// TIA Portal V15.1 export
// export: Created 2024-05-17T05:39:00.2667194Z, ExportSetting WithDefaults, DisplayName Totally Integrated Automation Portal, DisplayVersion V15.1 Update 5, DisplayName TIA Portal Openness, DisplayVersion V15.1 Update 5, DisplayName SINAMICS Startdrive Advanced, DisplayVersion V15.1, DisplayName G130, G150, S120, S150, SINAMICS MV, S210, DisplayVersion V15.1, DisplayName G110M, G120, G120C, G120D, G120P, DisplayVersion V15.1, DisplayName STEP 7 Professional, DisplayVersion V15.1 Update 5, DisplayName STEP 7 Safety, DisplayVersion V15.1, DisplayName WinCC Professional, DisplayVersion V15.1 Update 5, DisplayName SIMATIC Visualization Architect, DisplayVersion V15.1
FUNCTION "209000NCP01AK" : Void   // FC254, FBD
TITLE = 209000NCP01AK
{ S7_Optimized_Access := 'FALSE' }
AUTHOR : VCC
NAME : LocFnc
VERSION : 0.1
// stored: AutoNumber false, IsIECCheckEnabled false, SetENOAutomatically False, UDAEnableTagReadback false
   VAR_OUTPUT
      O_AlarmA : Bool;   // Alarm A
      O_AlarmB : Bool;   // Alarm B
      O_AlarmC : Bool;   // Alarm C
      O_AlarmD : Bool;   // Alarm D
      O_AlarmABCondition : Bool;   // Alarms resetable
      H_IAnim : Word;   // For animation of icon
   END_VAR
BEGIN

REGION Network 1: **** --------------------- AK01 --------------------- ****
END_REGION

REGION Network 2: **** 2.2 Alarms - Alarm generation **** AK01E1QM1 - AE01 EG1 - Overload protection power supply 24VDC
   // AE01 EG1 - Overload protection power supply 24VDC
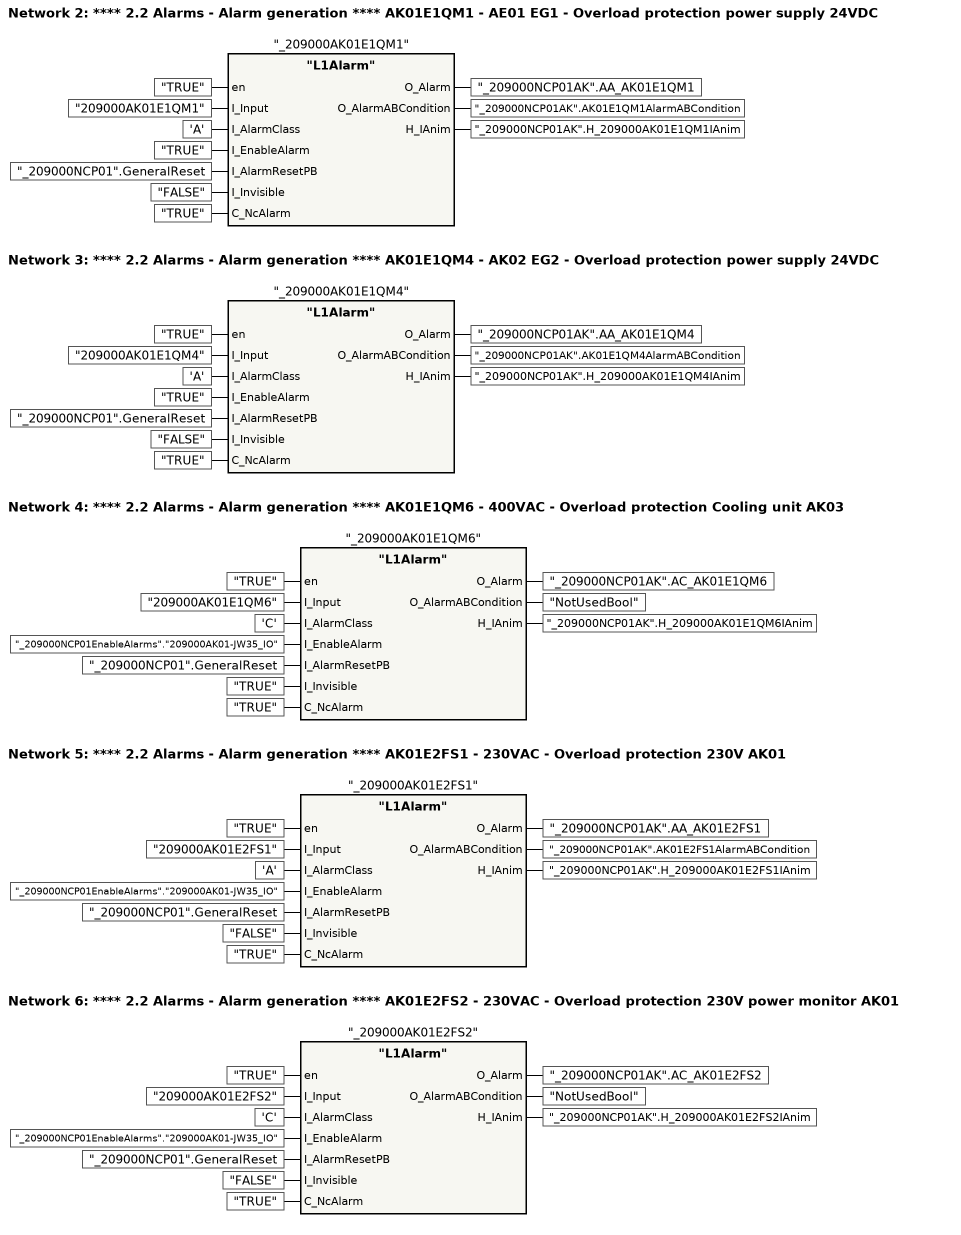
   IF "TRUE" THEN
       "_209000AK01E1QM1"(I_Input := "209000AK01E1QM1",   // "L1Alarm"
                          I_AlarmClass := 'A',
                          I_EnableAlarm := "TRUE",
                          I_AlarmResetPB := "_209000NCP01".GeneralReset,
                          I_Invisible := "FALSE",
                          C_NcAlarm := "TRUE",
                          O_Alarm => "_209000NCP01AK".AA_AK01E1QM1,
                          O_AlarmABCondition => "_209000NCP01AK".AK01E1QM1AlarmABCondition,
                          H_IAnim => "_209000NCP01AK".H_209000AK01E1QM1IAnim);
   END_IF;
END_REGION

REGION Network 3: **** 2.2 Alarms - Alarm generation **** AK01E1QM4 - AK02 EG2 - Overload protection power supply 24VDC
   // AK02 EG2 - Overload protection power supply 24VDC
   IF "TRUE" THEN
       "_209000AK01E1QM4"(I_Input := "209000AK01E1QM4",   // "L1Alarm"
                          I_AlarmClass := 'A',
                          I_EnableAlarm := "TRUE",
                          I_AlarmResetPB := "_209000NCP01".GeneralReset,
                          I_Invisible := "FALSE",
                          C_NcAlarm := "TRUE",
                          O_Alarm => "_209000NCP01AK".AA_AK01E1QM4,
                          O_AlarmABCondition => "_209000NCP01AK".AK01E1QM4AlarmABCondition,
                          H_IAnim => "_209000NCP01AK".H_209000AK01E1QM4IAnim);
   END_IF;
END_REGION

REGION Network 4: **** 2.2 Alarms - Alarm generation **** AK01E1QM6 - 400VAC - Overload protection Cooling unit AK03
   // 400VAC - Overload protection Cooling unit AK03
   IF "TRUE" THEN
       "_209000AK01E1QM6"(I_Input := "209000AK01E1QM6",   // "L1Alarm"
                          I_AlarmClass := 'C',
                          I_EnableAlarm := "_209000NCP01EnableAlarms"."209000AK01-JW35_IO",
                          I_AlarmResetPB := "_209000NCP01".GeneralReset,
                          I_Invisible := "TRUE",
                          C_NcAlarm := "TRUE",
                          O_Alarm => "_209000NCP01AK".AC_AK01E1QM6,
                          O_AlarmABCondition => "NotUsedBool",
                          H_IAnim => "_209000NCP01AK".H_209000AK01E1QM6IAnim);
   END_IF;
END_REGION

REGION Network 5: **** 2.2 Alarms - Alarm generation **** AK01E2FS1 - 230VAC - Overload protection 230V AK01
   // 230VAC - Overload protection 230V AK01
   IF "TRUE" THEN
       "_209000AK01E2FS1"(I_Input := "209000AK01E2FS1",   // "L1Alarm"
                          I_AlarmClass := 'A',
                          I_EnableAlarm := "_209000NCP01EnableAlarms"."209000AK01-JW35_IO",
                          I_AlarmResetPB := "_209000NCP01".GeneralReset,
                          I_Invisible := "FALSE",
                          C_NcAlarm := "TRUE",
                          O_Alarm => "_209000NCP01AK".AA_AK01E2FS1,
                          O_AlarmABCondition => "_209000NCP01AK".AK01E2FS1AlarmABCondition,
                          H_IAnim => "_209000NCP01AK".H_209000AK01E2FS1IAnim);
   END_IF;
END_REGION

REGION Network 6: **** 2.2 Alarms - Alarm generation **** AK01E2FS2 - 230VAC - Overload protection 230V power monitor AK01
   // 230VAC - Overload protection 230V power monitor AK01
   IF "TRUE" THEN
       "_209000AK01E2FS2"(I_Input := "209000AK01E2FS2",   // "L1Alarm"
                          I_AlarmClass := 'C',
                          I_EnableAlarm := "_209000NCP01EnableAlarms"."209000AK01-JW35_IO",
                          I_AlarmResetPB := "_209000NCP01".GeneralReset,
                          I_Invisible := "FALSE",
                          C_NcAlarm := "TRUE",
                          O_Alarm => "_209000NCP01AK".AC_AK01E2FS2,
                          O_AlarmABCondition => "NotUsedBool",
                          H_IAnim => "_209000NCP01AK".H_209000AK01E2FS2IAnim);
   END_IF;
END_REGION

REGION Network 7: **** 2.2 Alarms - Alarm generation **** AK01E2FS3 - 230VAC - Overload protection Socket + Light AK01-04
   // 230VAC - Overload protection Socket + Light AK01-04
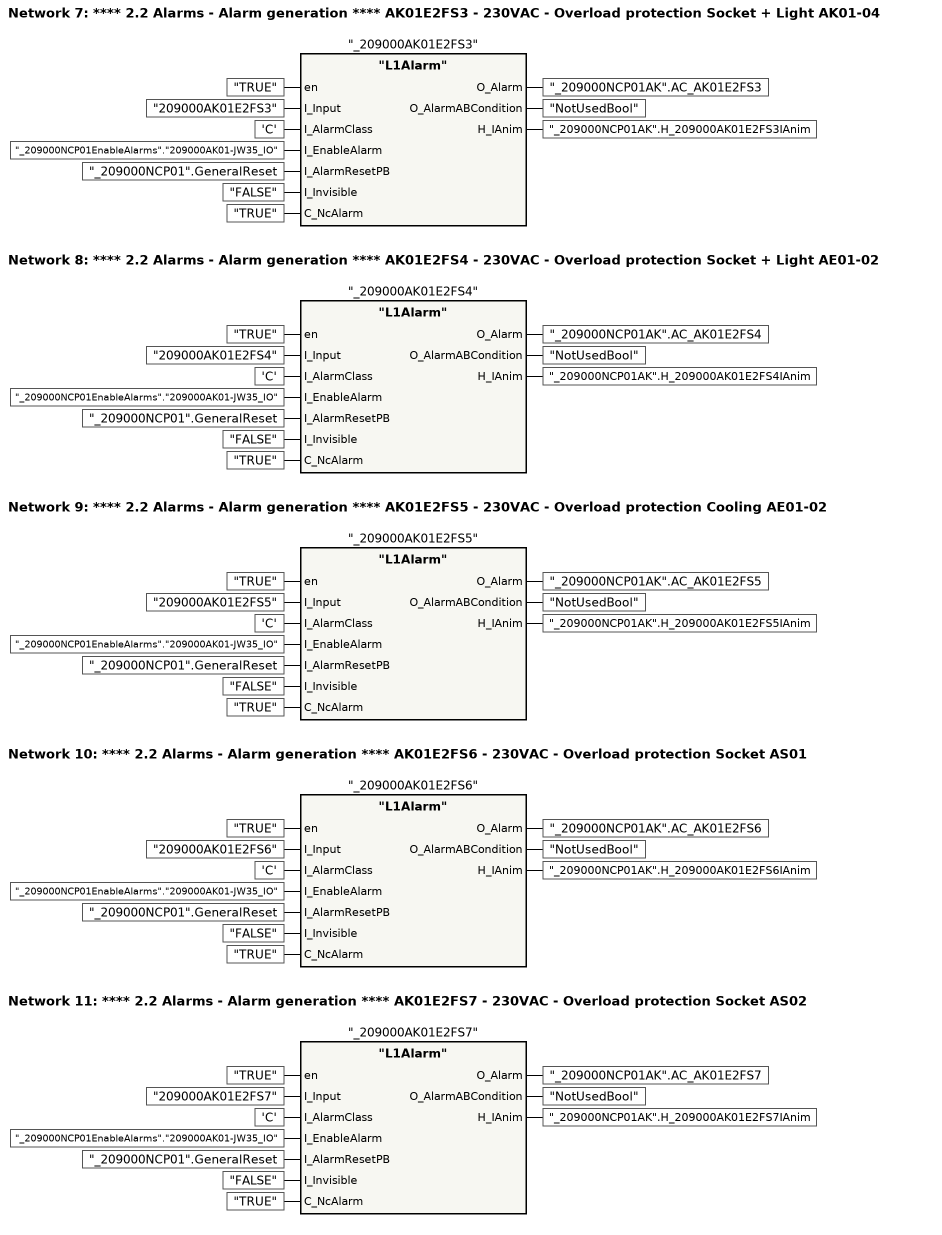
   IF "TRUE" THEN
       "_209000AK01E2FS3"(I_Input := "209000AK01E2FS3",   // "L1Alarm"
                          I_AlarmClass := 'C',
                          I_EnableAlarm := "_209000NCP01EnableAlarms"."209000AK01-JW35_IO",
                          I_AlarmResetPB := "_209000NCP01".GeneralReset,
                          I_Invisible := "FALSE",
                          C_NcAlarm := "TRUE",
                          O_Alarm => "_209000NCP01AK".AC_AK01E2FS3,
                          O_AlarmABCondition => "NotUsedBool",
                          H_IAnim => "_209000NCP01AK".H_209000AK01E2FS3IAnim);
   END_IF;
END_REGION

REGION Network 8: **** 2.2 Alarms - Alarm generation **** AK01E2FS4 - 230VAC - Overload protection Socket + Light AE01-02
   // 230VAC - Overload protection Socket + Light AE01-02
   IF "TRUE" THEN
       "_209000AK01E2FS4"(I_Input := "209000AK01E2FS4",   // "L1Alarm"
                          I_AlarmClass := 'C',
                          I_EnableAlarm := "_209000NCP01EnableAlarms"."209000AK01-JW35_IO",
                          I_AlarmResetPB := "_209000NCP01".GeneralReset,
                          I_Invisible := "FALSE",
                          C_NcAlarm := "TRUE",
                          O_Alarm => "_209000NCP01AK".AC_AK01E2FS4,
                          O_AlarmABCondition => "NotUsedBool",
                          H_IAnim => "_209000NCP01AK".H_209000AK01E2FS4IAnim);
   END_IF;
END_REGION

REGION Network 9: **** 2.2 Alarms - Alarm generation **** AK01E2FS5 - 230VAC - Overload protection Cooling AE01-02
   // 230VAC - Overload protection Cooling AE01-02
   IF "TRUE" THEN
       "_209000AK01E2FS5"(I_Input := "209000AK01E2FS5",   // "L1Alarm"
                          I_AlarmClass := 'C',
                          I_EnableAlarm := "_209000NCP01EnableAlarms"."209000AK01-JW35_IO",
                          I_AlarmResetPB := "_209000NCP01".GeneralReset,
                          I_Invisible := "FALSE",
                          C_NcAlarm := "TRUE",
                          O_Alarm => "_209000NCP01AK".AC_AK01E2FS5,
                          O_AlarmABCondition => "NotUsedBool",
                          H_IAnim => "_209000NCP01AK".H_209000AK01E2FS5IAnim);
   END_IF;
END_REGION

REGION Network 10: **** 2.2 Alarms - Alarm generation **** AK01E2FS6 - 230VAC - Overload protection Socket AS01
   // 230VAC - Overload protection Socket AS01
   IF "TRUE" THEN
       "_209000AK01E2FS6"(I_Input := "209000AK01E2FS6",   // "L1Alarm"
                          I_AlarmClass := 'C',
                          I_EnableAlarm := "_209000NCP01EnableAlarms"."209000AK01-JW35_IO",
                          I_AlarmResetPB := "_209000NCP01".GeneralReset,
                          I_Invisible := "FALSE",
                          C_NcAlarm := "TRUE",
                          O_Alarm => "_209000NCP01AK".AC_AK01E2FS6,
                          O_AlarmABCondition => "NotUsedBool",
                          H_IAnim => "_209000NCP01AK".H_209000AK01E2FS6IAnim);
   END_IF;
END_REGION

REGION Network 11: **** 2.2 Alarms - Alarm generation **** AK01E2FS7 - 230VAC - Overload protection Socket AS02
   // 230VAC - Overload protection Socket AS02
   IF "TRUE" THEN
       "_209000AK01E2FS7"(I_Input := "209000AK01E2FS7",   // "L1Alarm"
                          I_AlarmClass := 'C',
                          I_EnableAlarm := "_209000NCP01EnableAlarms"."209000AK01-JW35_IO",
                          I_AlarmResetPB := "_209000NCP01".GeneralReset,
                          I_Invisible := "FALSE",
                          C_NcAlarm := "TRUE",
                          O_Alarm => "_209000NCP01AK".AC_AK01E2FS7,
                          O_AlarmABCondition => "NotUsedBool",
                          H_IAnim => "_209000NCP01AK".H_209000AK01E2FS7IAnim);
   END_IF;
END_REGION

REGION Network 12: **** 2.2 Alarms - Alarm generation **** AK01E1FV1 - Surge protection 400VAC AK01 NOK
   // Surge protection 400VAC AK01 NOK
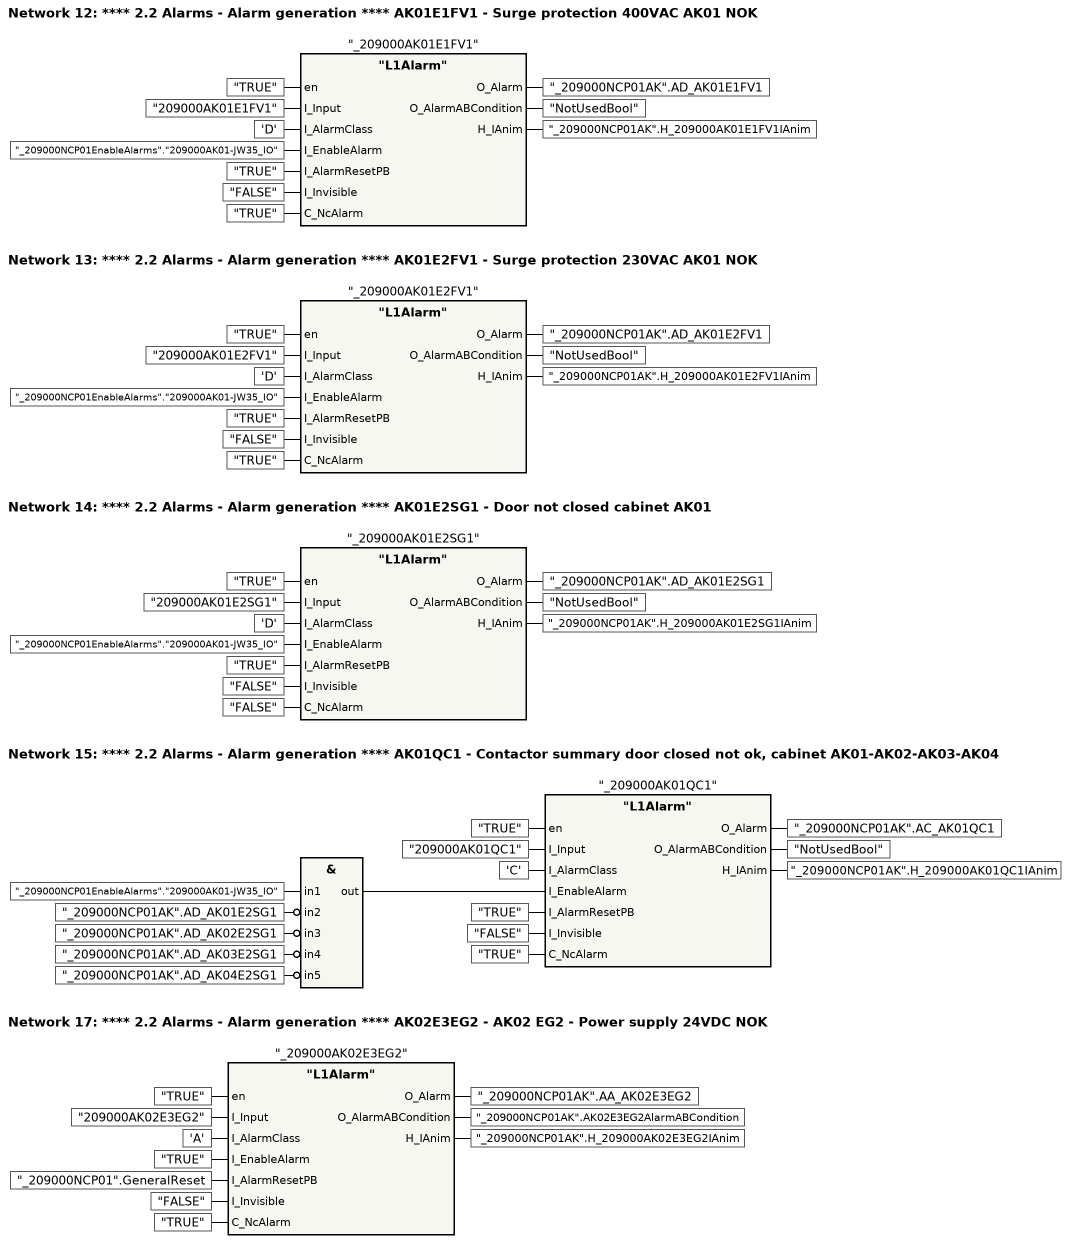
   IF "TRUE" THEN
       "_209000AK01E1FV1"(I_Input := "209000AK01E1FV1",   // "L1Alarm"
                          I_AlarmClass := 'D',
                          I_EnableAlarm := "_209000NCP01EnableAlarms"."209000AK01-JW35_IO",
                          I_AlarmResetPB := "TRUE",
                          I_Invisible := "FALSE",
                          C_NcAlarm := "TRUE",
                          O_Alarm => "_209000NCP01AK".AD_AK01E1FV1,
                          O_AlarmABCondition => "NotUsedBool",
                          H_IAnim => "_209000NCP01AK".H_209000AK01E1FV1IAnim);
   END_IF;
END_REGION

REGION Network 13: **** 2.2 Alarms - Alarm generation **** AK01E2FV1 - Surge protection 230VAC AK01 NOK
   // Surge protection 230VAC AK01 NOK
   IF "TRUE" THEN
       "_209000AK01E2FV1"(I_Input := "209000AK01E2FV1",   // "L1Alarm"
                          I_AlarmClass := 'D',
                          I_EnableAlarm := "_209000NCP01EnableAlarms"."209000AK01-JW35_IO",
                          I_AlarmResetPB := "TRUE",
                          I_Invisible := "FALSE",
                          C_NcAlarm := "TRUE",
                          O_Alarm => "_209000NCP01AK".AD_AK01E2FV1,
                          O_AlarmABCondition => "NotUsedBool",
                          H_IAnim => "_209000NCP01AK".H_209000AK01E2FV1IAnim);
   END_IF;
END_REGION

REGION Network 14: **** 2.2 Alarms - Alarm generation **** AK01E2SG1 - Door not closed cabinet AK01
   // Door not closed cabinet AK01
   IF "TRUE" THEN
       "_209000AK01E2SG1"(I_Input := "209000AK01E2SG1",   // "L1Alarm"
                          I_AlarmClass := 'D',
                          I_EnableAlarm := "_209000NCP01EnableAlarms"."209000AK01-JW35_IO",
                          I_AlarmResetPB := "TRUE",
                          I_Invisible := "FALSE",
                          C_NcAlarm := "FALSE",
                          O_Alarm => "_209000NCP01AK".AD_AK01E2SG1,
                          O_AlarmABCondition => "NotUsedBool",
                          H_IAnim => "_209000NCP01AK".H_209000AK01E2SG1IAnim);
   END_IF;
END_REGION

REGION Network 15: **** 2.2 Alarms - Alarm generation **** AK01QC1 - Contactor summary door closed not ok, cabinet AK01-AK02-AK03-AK04
   // Contactor summary door closed not ok, cabinet AK01-AK02-AK03-AK04
   IF "TRUE" THEN
       "_209000AK01QC1"(I_Input := "209000AK01QC1",   // "L1Alarm"
                        I_AlarmClass := 'C',
                        I_EnableAlarm := "_209000NCP01EnableAlarms"."209000AK01-JW35_IO" AND NOT "_209000NCP01AK".AD_AK01E2SG1 AND NOT "_209000NCP01AK".AD_AK02E2SG1 AND NOT "_209000NCP01AK".AD_AK03E2SG1 AND NOT "_209000NCP01AK".AD_AK04E2SG1,
                        I_AlarmResetPB := "TRUE",
                        I_Invisible := "FALSE",
                        C_NcAlarm := "TRUE",
                        O_Alarm => "_209000NCP01AK".AC_AK01QC1,
                        O_AlarmABCondition => "NotUsedBool",
                        H_IAnim => "_209000NCP01AK".H_209000AK01QC1IAnim);
   END_IF;
END_REGION

REGION Network 16: **** --------------------- AK02 --------------------- ****
END_REGION

REGION Network 17: **** 2.2 Alarms - Alarm generation **** AK02E3EG2 - AK02 EG2 - Power supply 24VDC NOK
   // AK02 EG2 - Power supply 24VDC NOK
   IF "TRUE" THEN
       "_209000AK02E3EG2"(I_Input := "209000AK02E3EG2",   // "L1Alarm"
                          I_AlarmClass := 'A',
                          I_EnableAlarm := "TRUE",
                          I_AlarmResetPB := "_209000NCP01".GeneralReset,
                          I_Invisible := "FALSE",
                          C_NcAlarm := "TRUE",
                          O_Alarm => "_209000NCP01AK".AA_AK02E3EG2,
                          O_AlarmABCondition => "_209000NCP01AK".AK02E3EG2AlarmABCondition,
                          H_IAnim => "_209000NCP01AK".H_209000AK02E3EG2IAnim);
   END_IF;
END_REGION

REGION Network 18: **** 2.2 Alarms - Alarm generation **** AK02E3FV2 - AK02 EG2 - Surge protection 24VDC NOK
   // AK02 EG2 - Surge protection 24VDC NOK
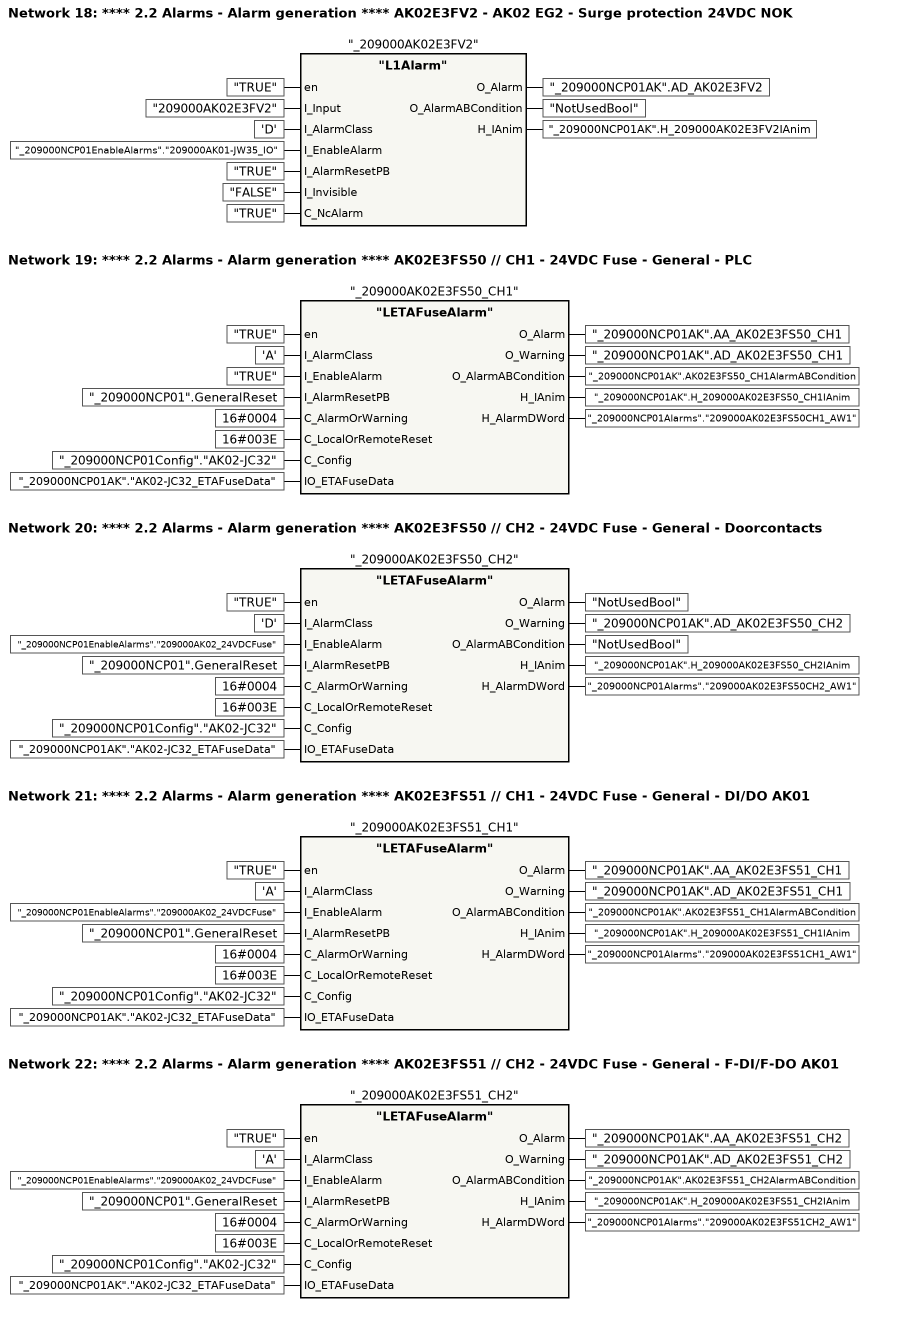
   IF "TRUE" THEN
       "_209000AK02E3FV2"(I_Input := "209000AK02E3FV2",   // "L1Alarm"
                          I_AlarmClass := 'D',
                          I_EnableAlarm := "_209000NCP01EnableAlarms"."209000AK01-JW35_IO",
                          I_AlarmResetPB := "TRUE",
                          I_Invisible := "FALSE",
                          C_NcAlarm := "TRUE",
                          O_Alarm => "_209000NCP01AK".AD_AK02E3FV2,
                          O_AlarmABCondition => "NotUsedBool",
                          H_IAnim => "_209000NCP01AK".H_209000AK02E3FV2IAnim);
   END_IF;
END_REGION

REGION Network 19: **** 2.2 Alarms - Alarm generation **** AK02E3FS50 // CH1 - 24VDC Fuse - General - PLC
   // 24VDC Fuse - General - PLC
   IF "TRUE" THEN
       "_209000AK02E3FS50_CH1"(I_AlarmClass := 'A',   // "LETAFuseAlarm"
                               I_EnableAlarm := "TRUE",
                               I_AlarmResetPB := "_209000NCP01".GeneralReset,
                               C_AlarmOrWarning := 16#0004,
                               C_LocalOrRemoteReset := 16#003E,
                               C_Config := "_209000NCP01Config"."AK02-JC32",
                               IO_ETAFuseData := "_209000NCP01AK"."AK02-JC32_ETAFuseData",
                               O_Alarm => "_209000NCP01AK".AA_AK02E3FS50_CH1,
                               O_Warning => "_209000NCP01AK".AD_AK02E3FS50_CH1,
                               O_AlarmABCondition => "_209000NCP01AK".AK02E3FS50_CH1AlarmABCondition,
                               H_IAnim => "_209000NCP01AK".H_209000AK02E3FS50_CH1IAnim,
                               H_AlarmDWord => "_209000NCP01Alarms"."209000AK02E3FS50CH1_AW1");
   END_IF;
END_REGION

REGION Network 20: **** 2.2 Alarms - Alarm generation **** AK02E3FS50 // CH2 - 24VDC Fuse - General - Doorcontacts
   // 24VDC Fuse - General - Doorcontacts
   IF "TRUE" THEN
       "_209000AK02E3FS50_CH2"(I_AlarmClass := 'D',   // "LETAFuseAlarm"
                               I_EnableAlarm := "_209000NCP01EnableAlarms"."209000AK02_24VDCFuse",
                               I_AlarmResetPB := "_209000NCP01".GeneralReset,
                               C_AlarmOrWarning := 16#0004,
                               C_LocalOrRemoteReset := 16#003E,
                               C_Config := "_209000NCP01Config"."AK02-JC32",
                               IO_ETAFuseData := "_209000NCP01AK"."AK02-JC32_ETAFuseData",
                               O_Alarm => "NotUsedBool",
                               O_Warning => "_209000NCP01AK".AD_AK02E3FS50_CH2,
                               O_AlarmABCondition => "NotUsedBool",
                               H_IAnim => "_209000NCP01AK".H_209000AK02E3FS50_CH2IAnim,
                               H_AlarmDWord => "_209000NCP01Alarms"."209000AK02E3FS50CH2_AW1");
   END_IF;
END_REGION

REGION Network 21: **** 2.2 Alarms - Alarm generation **** AK02E3FS51 // CH1 - 24VDC Fuse - General - DI/DO AK01
   // 24VDC Fuse - General - DI/DO AK01
   IF "TRUE" THEN
       "_209000AK02E3FS51_CH1"(I_AlarmClass := 'A',   // "LETAFuseAlarm"
                               I_EnableAlarm := "_209000NCP01EnableAlarms"."209000AK02_24VDCFuse",
                               I_AlarmResetPB := "_209000NCP01".GeneralReset,
                               C_AlarmOrWarning := 16#0004,
                               C_LocalOrRemoteReset := 16#003E,
                               C_Config := "_209000NCP01Config"."AK02-JC32",
                               IO_ETAFuseData := "_209000NCP01AK"."AK02-JC32_ETAFuseData",
                               O_Alarm => "_209000NCP01AK".AA_AK02E3FS51_CH1,
                               O_Warning => "_209000NCP01AK".AD_AK02E3FS51_CH1,
                               O_AlarmABCondition => "_209000NCP01AK".AK02E3FS51_CH1AlarmABCondition,
                               H_IAnim => "_209000NCP01AK".H_209000AK02E3FS51_CH1IAnim,
                               H_AlarmDWord => "_209000NCP01Alarms"."209000AK02E3FS51CH1_AW1");
   END_IF;
END_REGION

REGION Network 22: **** 2.2 Alarms - Alarm generation **** AK02E3FS51 // CH2 - 24VDC Fuse - General - F-DI/F-DO AK01
   // 24VDC Fuse - General - F-DI/F-DO AK01
   IF "TRUE" THEN
       "_209000AK02E3FS51_CH2"(I_AlarmClass := 'A',   // "LETAFuseAlarm"
                               I_EnableAlarm := "_209000NCP01EnableAlarms"."209000AK02_24VDCFuse",
                               I_AlarmResetPB := "_209000NCP01".GeneralReset,
                               C_AlarmOrWarning := 16#0004,
                               C_LocalOrRemoteReset := 16#003E,
                               C_Config := "_209000NCP01Config"."AK02-JC32",
                               IO_ETAFuseData := "_209000NCP01AK"."AK02-JC32_ETAFuseData",
                               O_Alarm => "_209000NCP01AK".AA_AK02E3FS51_CH2,
                               O_Warning => "_209000NCP01AK".AD_AK02E3FS51_CH2,
                               O_AlarmABCondition => "_209000NCP01AK".AK02E3FS51_CH2AlarmABCondition,
                               H_IAnim => "_209000NCP01AK".H_209000AK02E3FS51_CH2IAnim,
                               H_AlarmDWord => "_209000NCP01Alarms"."209000AK02E3FS51CH2_AW1");
   END_IF;
END_REGION

REGION Network 23: **** 2.2 Alarms - Alarm generation **** AK02E3FS52 // CH1 - 24VDC Fuse - General - DI/DO AK03
   // 24VDC Fuse - General - DI/DO AK03
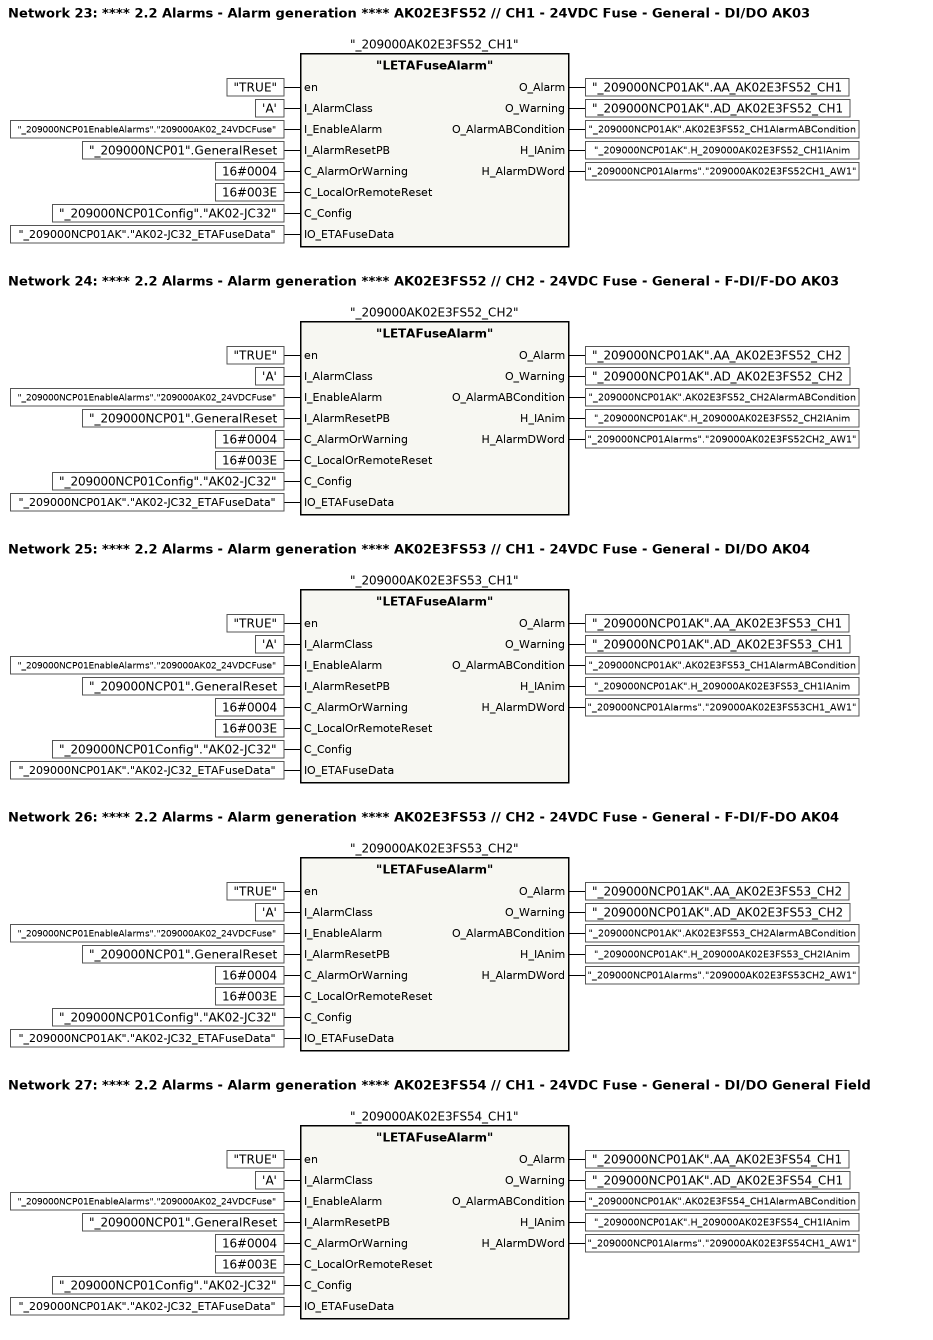
   IF "TRUE" THEN
       "_209000AK02E3FS52_CH1"(I_AlarmClass := 'A',   // "LETAFuseAlarm"
                               I_EnableAlarm := "_209000NCP01EnableAlarms"."209000AK02_24VDCFuse",
                               I_AlarmResetPB := "_209000NCP01".GeneralReset,
                               C_AlarmOrWarning := 16#0004,
                               C_LocalOrRemoteReset := 16#003E,
                               C_Config := "_209000NCP01Config"."AK02-JC32",
                               IO_ETAFuseData := "_209000NCP01AK"."AK02-JC32_ETAFuseData",
                               O_Alarm => "_209000NCP01AK".AA_AK02E3FS52_CH1,
                               O_Warning => "_209000NCP01AK".AD_AK02E3FS52_CH1,
                               O_AlarmABCondition => "_209000NCP01AK".AK02E3FS52_CH1AlarmABCondition,
                               H_IAnim => "_209000NCP01AK".H_209000AK02E3FS52_CH1IAnim,
                               H_AlarmDWord => "_209000NCP01Alarms"."209000AK02E3FS52CH1_AW1");
   END_IF;
END_REGION

REGION Network 24: **** 2.2 Alarms - Alarm generation **** AK02E3FS52 // CH2 - 24VDC Fuse - General - F-DI/F-DO AK03
   // 24VDC Fuse - General - F-DI/F-DO AK03
   IF "TRUE" THEN
       "_209000AK02E3FS52_CH2"(I_AlarmClass := 'A',   // "LETAFuseAlarm"
                               I_EnableAlarm := "_209000NCP01EnableAlarms"."209000AK02_24VDCFuse",
                               I_AlarmResetPB := "_209000NCP01".GeneralReset,
                               C_AlarmOrWarning := 16#0004,
                               C_LocalOrRemoteReset := 16#003E,
                               C_Config := "_209000NCP01Config"."AK02-JC32",
                               IO_ETAFuseData := "_209000NCP01AK"."AK02-JC32_ETAFuseData",
                               O_Alarm => "_209000NCP01AK".AA_AK02E3FS52_CH2,
                               O_Warning => "_209000NCP01AK".AD_AK02E3FS52_CH2,
                               O_AlarmABCondition => "_209000NCP01AK".AK02E3FS52_CH2AlarmABCondition,
                               H_IAnim => "_209000NCP01AK".H_209000AK02E3FS52_CH2IAnim,
                               H_AlarmDWord => "_209000NCP01Alarms"."209000AK02E3FS52CH2_AW1");
   END_IF;
END_REGION

REGION Network 25: **** 2.2 Alarms - Alarm generation **** AK02E3FS53 // CH1 - 24VDC Fuse - General - DI/DO AK04
   // 24VDC Fuse - General - DI/DO AK04
   IF "TRUE" THEN
       "_209000AK02E3FS53_CH1"(I_AlarmClass := 'A',   // "LETAFuseAlarm"
                               I_EnableAlarm := "_209000NCP01EnableAlarms"."209000AK02_24VDCFuse",
                               I_AlarmResetPB := "_209000NCP01".GeneralReset,
                               C_AlarmOrWarning := 16#0004,
                               C_LocalOrRemoteReset := 16#003E,
                               C_Config := "_209000NCP01Config"."AK02-JC32",
                               IO_ETAFuseData := "_209000NCP01AK"."AK02-JC32_ETAFuseData",
                               O_Alarm => "_209000NCP01AK".AA_AK02E3FS53_CH1,
                               O_Warning => "_209000NCP01AK".AD_AK02E3FS53_CH1,
                               O_AlarmABCondition => "_209000NCP01AK".AK02E3FS53_CH1AlarmABCondition,
                               H_IAnim => "_209000NCP01AK".H_209000AK02E3FS53_CH1IAnim,
                               H_AlarmDWord => "_209000NCP01Alarms"."209000AK02E3FS53CH1_AW1");
   END_IF;
END_REGION

REGION Network 26: **** 2.2 Alarms - Alarm generation **** AK02E3FS53 // CH2 - 24VDC Fuse - General - F-DI/F-DO AK04
   // 24VDC Fuse - General - F-DI/F-DO AK04
   IF "TRUE" THEN
       "_209000AK02E3FS53_CH2"(I_AlarmClass := 'A',   // "LETAFuseAlarm"
                               I_EnableAlarm := "_209000NCP01EnableAlarms"."209000AK02_24VDCFuse",
                               I_AlarmResetPB := "_209000NCP01".GeneralReset,
                               C_AlarmOrWarning := 16#0004,
                               C_LocalOrRemoteReset := 16#003E,
                               C_Config := "_209000NCP01Config"."AK02-JC32",
                               IO_ETAFuseData := "_209000NCP01AK"."AK02-JC32_ETAFuseData",
                               O_Alarm => "_209000NCP01AK".AA_AK02E3FS53_CH2,
                               O_Warning => "_209000NCP01AK".AD_AK02E3FS53_CH2,
                               O_AlarmABCondition => "_209000NCP01AK".AK02E3FS53_CH2AlarmABCondition,
                               H_IAnim => "_209000NCP01AK".H_209000AK02E3FS53_CH2IAnim,
                               H_AlarmDWord => "_209000NCP01Alarms"."209000AK02E3FS53CH2_AW1");
   END_IF;
END_REGION

REGION Network 27: **** 2.2 Alarms - Alarm generation **** AK02E3FS54 // CH1 - 24VDC Fuse - General - DI/DO General Field
   // 24VDC Fuse - General - DI/DO General Field
   IF "TRUE" THEN
       "_209000AK02E3FS54_CH1"(I_AlarmClass := 'A',   // "LETAFuseAlarm"
                               I_EnableAlarm := "_209000NCP01EnableAlarms"."209000AK02_24VDCFuse",
                               I_AlarmResetPB := "_209000NCP01".GeneralReset,
                               C_AlarmOrWarning := 16#0004,
                               C_LocalOrRemoteReset := 16#003E,
                               C_Config := "_209000NCP01Config"."AK02-JC32",
                               IO_ETAFuseData := "_209000NCP01AK"."AK02-JC32_ETAFuseData",
                               O_Alarm => "_209000NCP01AK".AA_AK02E3FS54_CH1,
                               O_Warning => "_209000NCP01AK".AD_AK02E3FS54_CH1,
                               O_AlarmABCondition => "_209000NCP01AK".AK02E3FS54_CH1AlarmABCondition,
                               H_IAnim => "_209000NCP01AK".H_209000AK02E3FS54_CH1IAnim,
                               H_AlarmDWord => "_209000NCP01Alarms"."209000AK02E3FS54CH1_AW1");
   END_IF;
END_REGION

REGION Network 28: **** 2.2 Alarms - Alarm generation **** AK02E3FS54 // CH2 - 24VDC Fuse - General - F-DI/F-DO General Field
   // 24VDC Fuse - General - F-DI/F-DO General Field
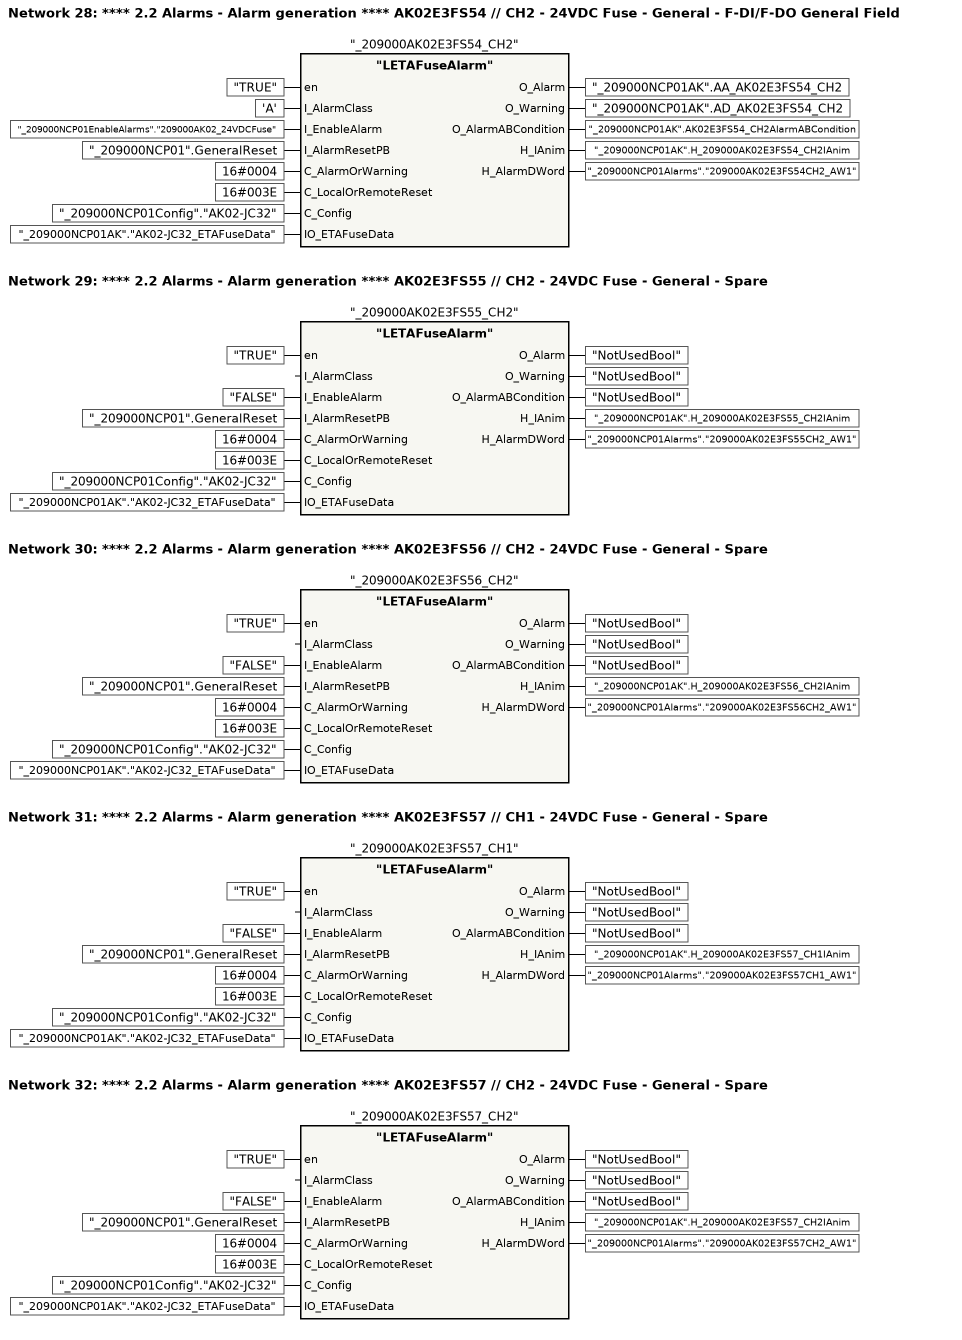
   IF "TRUE" THEN
       "_209000AK02E3FS54_CH2"(I_AlarmClass := 'A',   // "LETAFuseAlarm"
                               I_EnableAlarm := "_209000NCP01EnableAlarms"."209000AK02_24VDCFuse",
                               I_AlarmResetPB := "_209000NCP01".GeneralReset,
                               C_AlarmOrWarning := 16#0004,
                               C_LocalOrRemoteReset := 16#003E,
                               C_Config := "_209000NCP01Config"."AK02-JC32",
                               IO_ETAFuseData := "_209000NCP01AK"."AK02-JC32_ETAFuseData",
                               O_Alarm => "_209000NCP01AK".AA_AK02E3FS54_CH2,
                               O_Warning => "_209000NCP01AK".AD_AK02E3FS54_CH2,
                               O_AlarmABCondition => "_209000NCP01AK".AK02E3FS54_CH2AlarmABCondition,
                               H_IAnim => "_209000NCP01AK".H_209000AK02E3FS54_CH2IAnim,
                               H_AlarmDWord => "_209000NCP01Alarms"."209000AK02E3FS54CH2_AW1");
   END_IF;
END_REGION

REGION Network 29: **** 2.2 Alarms - Alarm generation **** AK02E3FS55 // CH2 - 24VDC Fuse - General - Spare
   // 24VDC Fuse - General - Spare
   IF "TRUE" THEN
       "_209000AK02E3FS55_CH2"(I_EnableAlarm := "FALSE",   // "LETAFuseAlarm"
                               I_AlarmResetPB := "_209000NCP01".GeneralReset,
                               C_AlarmOrWarning := 16#0004,
                               C_LocalOrRemoteReset := 16#003E,
                               C_Config := "_209000NCP01Config"."AK02-JC32",
                               IO_ETAFuseData := "_209000NCP01AK"."AK02-JC32_ETAFuseData",
                               O_Alarm => "NotUsedBool",
                               O_Warning => "NotUsedBool",
                               O_AlarmABCondition => "NotUsedBool",
                               H_IAnim => "_209000NCP01AK".H_209000AK02E3FS55_CH2IAnim,
                               H_AlarmDWord => "_209000NCP01Alarms"."209000AK02E3FS55CH2_AW1");
   END_IF;
END_REGION

REGION Network 30: **** 2.2 Alarms - Alarm generation **** AK02E3FS56 // CH2 - 24VDC Fuse - General - Spare
   // 24VDC Fuse - General - Spare
   IF "TRUE" THEN
       "_209000AK02E3FS56_CH2"(I_EnableAlarm := "FALSE",   // "LETAFuseAlarm"
                               I_AlarmResetPB := "_209000NCP01".GeneralReset,
                               C_AlarmOrWarning := 16#0004,
                               C_LocalOrRemoteReset := 16#003E,
                               C_Config := "_209000NCP01Config"."AK02-JC32",
                               IO_ETAFuseData := "_209000NCP01AK"."AK02-JC32_ETAFuseData",
                               O_Alarm => "NotUsedBool",
                               O_Warning => "NotUsedBool",
                               O_AlarmABCondition => "NotUsedBool",
                               H_IAnim => "_209000NCP01AK".H_209000AK02E3FS56_CH2IAnim,
                               H_AlarmDWord => "_209000NCP01Alarms"."209000AK02E3FS56CH2_AW1");
   END_IF;
END_REGION

REGION Network 31: **** 2.2 Alarms - Alarm generation **** AK02E3FS57 // CH1 - 24VDC Fuse - General - Spare
   // 24VDC Fuse - General - Spare
   IF "TRUE" THEN
       "_209000AK02E3FS57_CH1"(I_EnableAlarm := "FALSE",   // "LETAFuseAlarm"
                               I_AlarmResetPB := "_209000NCP01".GeneralReset,
                               C_AlarmOrWarning := 16#0004,
                               C_LocalOrRemoteReset := 16#003E,
                               C_Config := "_209000NCP01Config"."AK02-JC32",
                               IO_ETAFuseData := "_209000NCP01AK"."AK02-JC32_ETAFuseData",
                               O_Alarm => "NotUsedBool",
                               O_Warning => "NotUsedBool",
                               O_AlarmABCondition => "NotUsedBool",
                               H_IAnim => "_209000NCP01AK".H_209000AK02E3FS57_CH1IAnim,
                               H_AlarmDWord => "_209000NCP01Alarms"."209000AK02E3FS57CH1_AW1");
   END_IF;
END_REGION

REGION Network 32: **** 2.2 Alarms - Alarm generation **** AK02E3FS57 // CH2 - 24VDC Fuse - General - Spare
   // 24VDC Fuse - General - Spare
   IF "TRUE" THEN
       "_209000AK02E3FS57_CH2"(I_EnableAlarm := "FALSE",   // "LETAFuseAlarm"
                               I_AlarmResetPB := "_209000NCP01".GeneralReset,
                               C_AlarmOrWarning := 16#0004,
                               C_LocalOrRemoteReset := 16#003E,
                               C_Config := "_209000NCP01Config"."AK02-JC32",
                               IO_ETAFuseData := "_209000NCP01AK"."AK02-JC32_ETAFuseData",
                               O_Alarm => "NotUsedBool",
                               O_Warning => "NotUsedBool",
                               O_AlarmABCondition => "NotUsedBool",
                               H_IAnim => "_209000NCP01AK".H_209000AK02E3FS57_CH2IAnim,
                               H_AlarmDWord => "_209000NCP01Alarms"."209000AK02E3FS57CH2_AW1");
   END_IF;
END_REGION

REGION Network 33: **** 2.2 Alarms - Alarm generation **** AK02E2SG1 - Door not closed cabinet AK02
   // Door not closed cabinet AK02
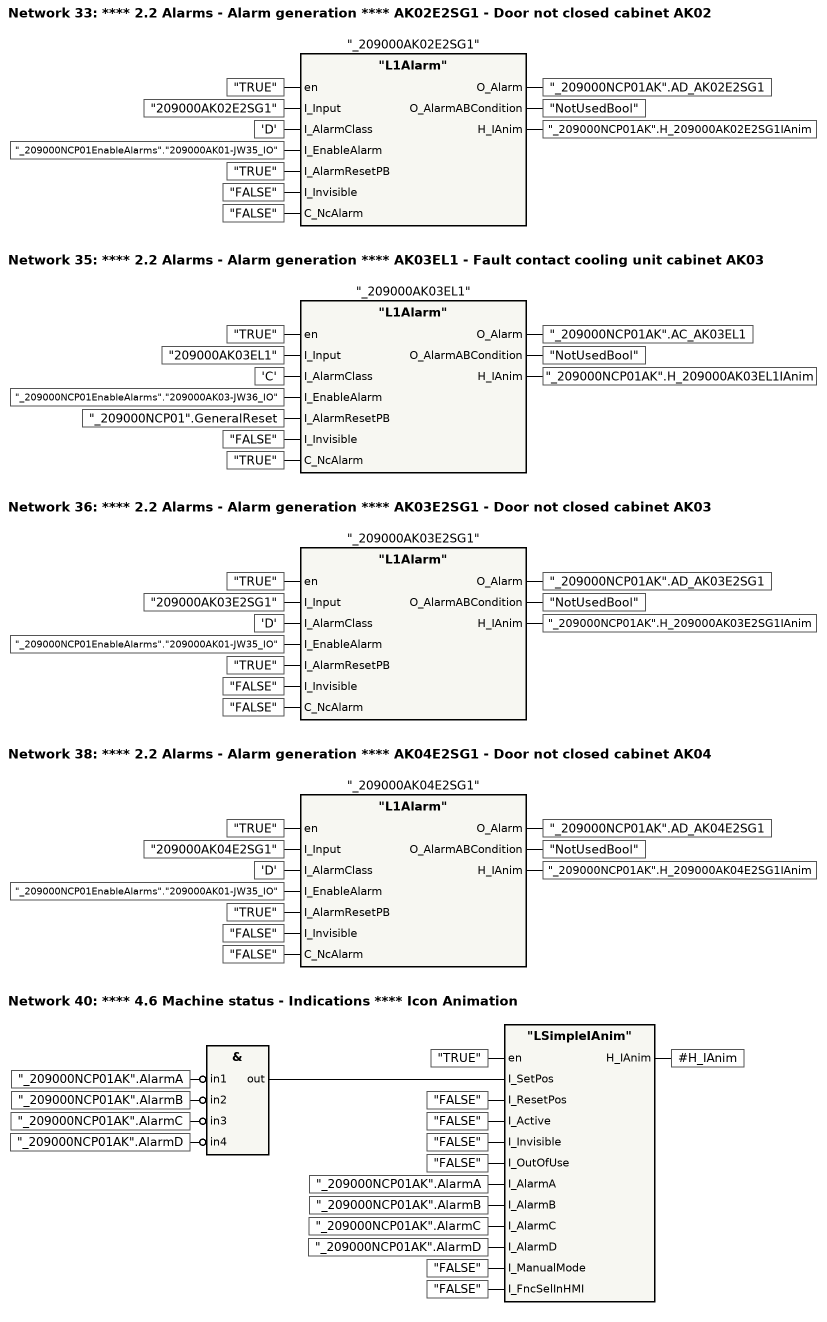
   IF "TRUE" THEN
       "_209000AK02E2SG1"(I_Input := "209000AK02E2SG1",   // "L1Alarm"
                          I_AlarmClass := 'D',
                          I_EnableAlarm := "_209000NCP01EnableAlarms"."209000AK01-JW35_IO",
                          I_AlarmResetPB := "TRUE",
                          I_Invisible := "FALSE",
                          C_NcAlarm := "FALSE",
                          O_Alarm => "_209000NCP01AK".AD_AK02E2SG1,
                          O_AlarmABCondition => "NotUsedBool",
                          H_IAnim => "_209000NCP01AK".H_209000AK02E2SG1IAnim);
   END_IF;
END_REGION

REGION Network 34: **** --------------------- AK03 --------------------- ****
END_REGION

REGION Network 35: **** 2.2 Alarms - Alarm generation **** AK03EL1 - Fault contact cooling unit cabinet AK03
   // Fault contact cooling unit cabinet AK03
   IF "TRUE" THEN
       "_209000AK03EL1"(I_Input := "209000AK03EL1",   // "L1Alarm"
                        I_AlarmClass := 'C',
                        I_EnableAlarm := "_209000NCP01EnableAlarms"."209000AK03-JW36_IO",
                        I_AlarmResetPB := "_209000NCP01".GeneralReset,
                        I_Invisible := "FALSE",
                        C_NcAlarm := "TRUE",
                        O_Alarm => "_209000NCP01AK".AC_AK03EL1,
                        O_AlarmABCondition => "NotUsedBool",
                        H_IAnim => "_209000NCP01AK".H_209000AK03EL1IAnim);
   END_IF;
END_REGION

REGION Network 36: **** 2.2 Alarms - Alarm generation **** AK03E2SG1 - Door not closed cabinet AK03
   // Door not closed cabinet AK03
   IF "TRUE" THEN
       "_209000AK03E2SG1"(I_Input := "209000AK03E2SG1",   // "L1Alarm"
                          I_AlarmClass := 'D',
                          I_EnableAlarm := "_209000NCP01EnableAlarms"."209000AK01-JW35_IO",
                          I_AlarmResetPB := "TRUE",
                          I_Invisible := "FALSE",
                          C_NcAlarm := "FALSE",
                          O_Alarm => "_209000NCP01AK".AD_AK03E2SG1,
                          O_AlarmABCondition => "NotUsedBool",
                          H_IAnim => "_209000NCP01AK".H_209000AK03E2SG1IAnim);
   END_IF;
END_REGION

REGION Network 37: **** --------------------- AK04 --------------------- ****
END_REGION

REGION Network 38: **** 2.2 Alarms - Alarm generation **** AK04E2SG1 - Door not closed cabinet AK04
   // Door not closed cabinet AK04
   IF "TRUE" THEN
       "_209000AK04E2SG1"(I_Input := "209000AK04E2SG1",   // "L1Alarm"
                          I_AlarmClass := 'D',
                          I_EnableAlarm := "_209000NCP01EnableAlarms"."209000AK01-JW35_IO",
                          I_AlarmResetPB := "TRUE",
                          I_Invisible := "FALSE",
                          C_NcAlarm := "FALSE",
                          O_Alarm => "_209000NCP01AK".AD_AK04E2SG1,
                          O_AlarmABCondition => "NotUsedBool",
                          H_IAnim => "_209000NCP01AK".H_209000AK04E2SG1IAnim);
   END_IF;
END_REGION

REGION Network 39: **** -------------------------------------------------- ****
END_REGION

REGION Network 40: **** 4.6 Machine status - Indications **** Icon Animation
   // Animation for icon
   IF "TRUE" THEN
       "LSimpleIAnim"(I_SetPos := NOT "_209000NCP01AK".AlarmA AND NOT "_209000NCP01AK".AlarmB AND NOT "_209000NCP01AK".AlarmC AND NOT "_209000NCP01AK".AlarmD,
                      I_ResetPos := "FALSE",
                      I_Active := "FALSE",
                      I_Invisible := "FALSE",
                      I_OutOfUse := "FALSE",
                      I_AlarmA := "_209000NCP01AK".AlarmA,
                      I_AlarmB := "_209000NCP01AK".AlarmB,
                      I_AlarmC := "_209000NCP01AK".AlarmC,
                      I_AlarmD := "_209000NCP01AK".AlarmD,
                      I_ManualMode := "FALSE",
                      I_FncSelInHMI := "FALSE",
                      H_IAnim => #H_IAnim);
   END_IF;
END_REGION

REGION Network 41: **** 4.6 - Machine status - Indications **** Animation
   // Animation
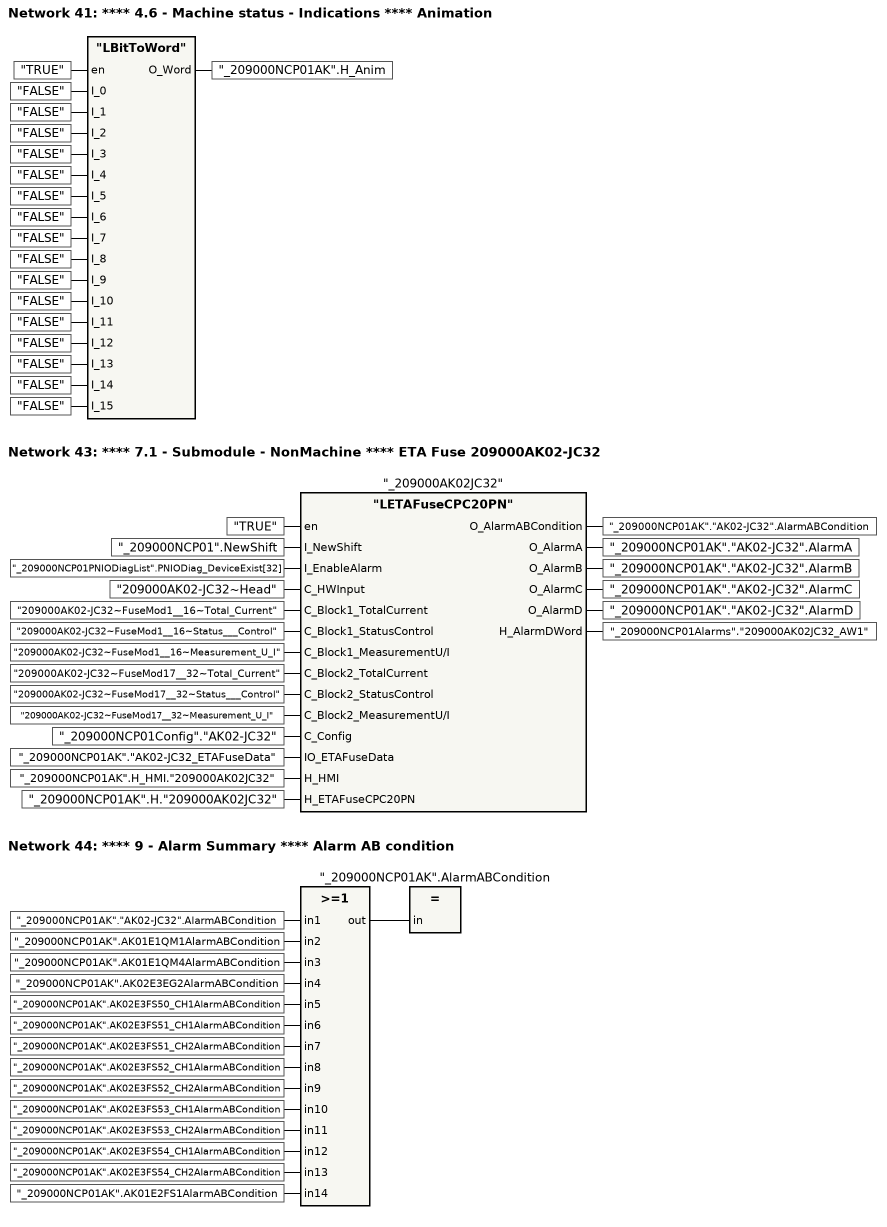
   IF "TRUE" THEN
       "LBitToWord"(I_0 := "FALSE",
                    I_1 := "FALSE",
                    I_2 := "FALSE",
                    I_3 := "FALSE",
                    I_4 := "FALSE",
                    I_5 := "FALSE",
                    I_6 := "FALSE",
                    I_7 := "FALSE",
                    I_8 := "FALSE",
                    I_9 := "FALSE",
                    I_10 := "FALSE",
                    I_11 := "FALSE",
                    I_12 := "FALSE",
                    I_13 := "FALSE",
                    I_14 := "FALSE",
                    I_15 := "FALSE",
                    O_Word => "_209000NCP01AK".H_Anim);
   END_IF;
END_REGION

NETWORK
TITLE = **** 4.6 - Machine Status - Indications **** Animation DB number
// DB number
      OPN   "_209000NCP01AK";
      L     DBNO;
      T     "_209000NCP01AK".H_DBnr;

REGION Network 43: **** 7.1 - Submodule - NonMachine **** ETA Fuse 209000AK02-JC32
   IF "TRUE" THEN
       "_209000AK02JC32"(I_NewShift := "_209000NCP01".NewShift,   // "LETAFuseCPC20PN"
                         I_EnableAlarm := "_209000NCP01PNIODiagList".PNIODiag_DeviceExist[32],
                         C_HWInput := "209000AK02-JC32~Head",
                         C_Block1_TotalCurrent := "209000AK02-JC32~FuseMod1__16~Total_Current",
                         C_Block1_StatusControl := "209000AK02-JC32~FuseMod1__16~Status___Control",
                         "C_Block1_MeasurementU/I" := "209000AK02-JC32~FuseMod1__16~Measurement_U_I",
                         C_Block2_TotalCurrent := "209000AK02-JC32~FuseMod17__32~Total_Current",
                         C_Block2_StatusControl := "209000AK02-JC32~FuseMod17__32~Status___Control",
                         "C_Block2_MeasurementU/I" := "209000AK02-JC32~FuseMod17__32~Measurement_U_I",
                         C_Config := "_209000NCP01Config"."AK02-JC32",
                         IO_ETAFuseData := "_209000NCP01AK"."AK02-JC32_ETAFuseData",
                         H_HMI := "_209000NCP01AK".H_HMI."209000AK02JC32",
                         H_ETAFuseCPC20PN := "_209000NCP01AK".H."209000AK02JC32",
                         O_AlarmABCondition => "_209000NCP01AK"."AK02-JC32".AlarmABCondition,
                         O_AlarmA => "_209000NCP01AK"."AK02-JC32".AlarmA,
                         O_AlarmB => "_209000NCP01AK"."AK02-JC32".AlarmB,
                         O_AlarmC => "_209000NCP01AK"."AK02-JC32".AlarmC,
                         O_AlarmD => "_209000NCP01AK"."AK02-JC32".AlarmD,
                         H_AlarmDWord => "_209000NCP01Alarms"."209000AK02JC32_AW1");
   END_IF;
END_REGION

REGION Network 44: **** 9 - Alarm Summary **** Alarm AB condition
   // Alarm AB condition
   "_209000NCP01AK".AlarmABCondition := "_209000NCP01AK"."AK02-JC32".AlarmABCondition OR "_209000NCP01AK".AK01E1QM1AlarmABCondition OR "_209000NCP01AK".AK01E1QM4AlarmABCondition OR "_209000NCP01AK".AK02E3EG2AlarmABCondition OR "_209000NCP01AK".AK02E3FS50_CH1AlarmABCondition OR "_209000NCP01AK".AK02E3FS51_CH1AlarmABCondition OR "_209000NCP01AK".AK02E3FS51_CH2AlarmABCondition OR "_209000NCP01AK".AK02E3FS52_CH1AlarmABCondition OR "_209000NCP01AK".AK02E3FS52_CH2AlarmABCondition OR "_209000NCP01AK".AK02E3FS53_CH1AlarmABCondition OR "_209000NCP01AK".AK02E3FS53_CH2AlarmABCondition OR "_209000NCP01AK".AK02E3FS54_CH1AlarmABCondition OR "_209000NCP01AK".AK02E3FS54_CH2AlarmABCondition OR "_209000NCP01AK".AK01E2FS1AlarmABCondition;
END_REGION

REGION Network 45: **** 9 - Alarm Summary **** Alarm A
   // Summary of alarms A
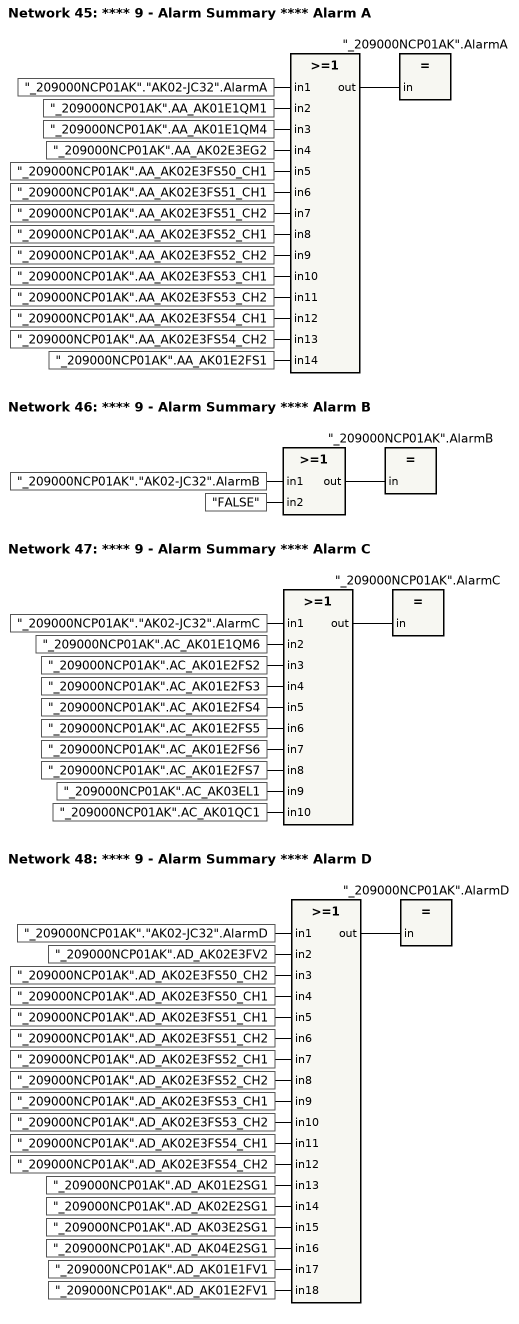
   "_209000NCP01AK".AlarmA := "_209000NCP01AK"."AK02-JC32".AlarmA OR "_209000NCP01AK".AA_AK01E1QM1 OR "_209000NCP01AK".AA_AK01E1QM4 OR "_209000NCP01AK".AA_AK02E3EG2 OR "_209000NCP01AK".AA_AK02E3FS50_CH1 OR "_209000NCP01AK".AA_AK02E3FS51_CH1 OR "_209000NCP01AK".AA_AK02E3FS51_CH2 OR "_209000NCP01AK".AA_AK02E3FS52_CH1 OR "_209000NCP01AK".AA_AK02E3FS52_CH2 OR "_209000NCP01AK".AA_AK02E3FS53_CH1 OR "_209000NCP01AK".AA_AK02E3FS53_CH2 OR "_209000NCP01AK".AA_AK02E3FS54_CH1 OR "_209000NCP01AK".AA_AK02E3FS54_CH2 OR "_209000NCP01AK".AA_AK01E2FS1;
END_REGION

REGION Network 46: **** 9 - Alarm Summary **** Alarm B
   // Summary of alarms B
   "_209000NCP01AK".AlarmB := "_209000NCP01AK"."AK02-JC32".AlarmB OR "FALSE";
END_REGION

REGION Network 47: **** 9 - Alarm Summary **** Alarm C
   // Summary of alarms C
   "_209000NCP01AK".AlarmC := "_209000NCP01AK"."AK02-JC32".AlarmC OR "_209000NCP01AK".AC_AK01E1QM6 OR "_209000NCP01AK".AC_AK01E2FS2 OR "_209000NCP01AK".AC_AK01E2FS3 OR "_209000NCP01AK".AC_AK01E2FS4 OR "_209000NCP01AK".AC_AK01E2FS5 OR "_209000NCP01AK".AC_AK01E2FS6 OR "_209000NCP01AK".AC_AK01E2FS7 OR "_209000NCP01AK".AC_AK03EL1 OR "_209000NCP01AK".AC_AK01QC1;
END_REGION

REGION Network 48: **** 9 - Alarm Summary **** Alarm D
   // Summary of alarms D
   "_209000NCP01AK".AlarmD := "_209000NCP01AK"."AK02-JC32".AlarmD OR "_209000NCP01AK".AD_AK02E3FV2 OR "_209000NCP01AK".AD_AK02E3FS50_CH2 OR "_209000NCP01AK".AD_AK02E3FS50_CH1 OR "_209000NCP01AK".AD_AK02E3FS51_CH1 OR "_209000NCP01AK".AD_AK02E3FS51_CH2 OR "_209000NCP01AK".AD_AK02E3FS52_CH1 OR "_209000NCP01AK".AD_AK02E3FS52_CH2 OR "_209000NCP01AK".AD_AK02E3FS53_CH1 OR "_209000NCP01AK".AD_AK02E3FS53_CH2 OR "_209000NCP01AK".AD_AK02E3FS54_CH1 OR "_209000NCP01AK".AD_AK02E3FS54_CH2 OR "_209000NCP01AK".AD_AK01E2SG1 OR "_209000NCP01AK".AD_AK02E2SG1 OR "_209000NCP01AK".AD_AK03E2SG1 OR "_209000NCP01AK".AD_AK04E2SG1 OR "_209000NCP01AK".AD_AK01E1FV1 OR "_209000NCP01AK".AD_AK01E2FV1;
END_REGION

REGION Network 49: **** 9.1 - Alarm Output **** Alarm AB condition
   // Alarm AB condition
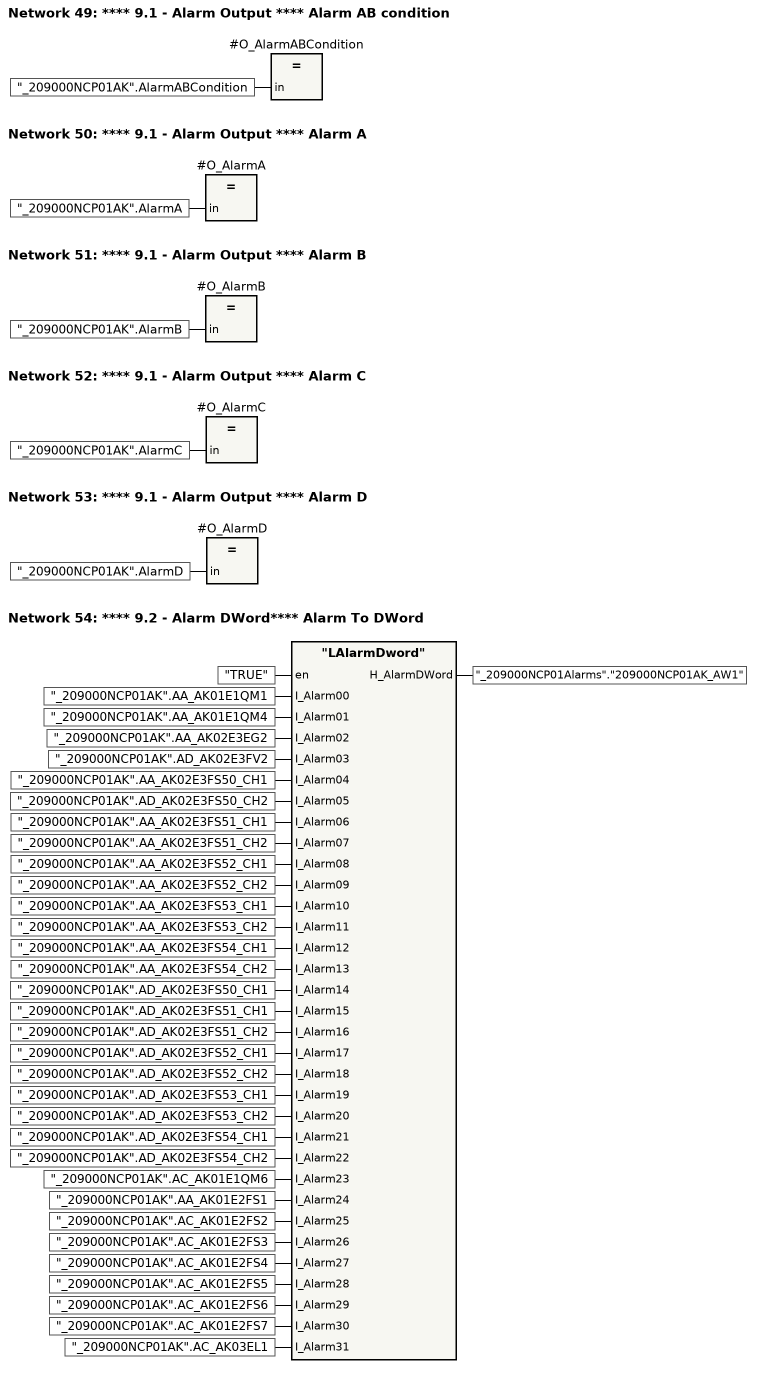
   #O_AlarmABCondition := "_209000NCP01AK".AlarmABCondition;
END_REGION

REGION Network 50: **** 9.1 - Alarm Output **** Alarm A
   // Summary of alarms A
   #O_AlarmA := "_209000NCP01AK".AlarmA;
END_REGION

REGION Network 51: **** 9.1 - Alarm Output **** Alarm B
   // Summary of alarms B
   #O_AlarmB := "_209000NCP01AK".AlarmB;
END_REGION

REGION Network 52: **** 9.1 - Alarm Output **** Alarm C
   // Summary of alarms C
   #O_AlarmC := "_209000NCP01AK".AlarmC;
END_REGION

REGION Network 53: **** 9.1 - Alarm Output **** Alarm D
   // Summary of alarms D
   #O_AlarmD := "_209000NCP01AK".AlarmD;
END_REGION

REGION Network 54: **** 9.2 - Alarm DWord**** Alarm To DWord
   // Alarm Word
   IF "TRUE" THEN
       "LAlarmDword"(I_Alarm00 := "_209000NCP01AK".AA_AK01E1QM1,
                     I_Alarm01 := "_209000NCP01AK".AA_AK01E1QM4,
                     I_Alarm02 := "_209000NCP01AK".AA_AK02E3EG2,
                     I_Alarm03 := "_209000NCP01AK".AD_AK02E3FV2,
                     I_Alarm04 := "_209000NCP01AK".AA_AK02E3FS50_CH1,
                     I_Alarm05 := "_209000NCP01AK".AD_AK02E3FS50_CH2,
                     I_Alarm06 := "_209000NCP01AK".AA_AK02E3FS51_CH1,
                     I_Alarm07 := "_209000NCP01AK".AA_AK02E3FS51_CH2,
                     I_Alarm08 := "_209000NCP01AK".AA_AK02E3FS52_CH1,
                     I_Alarm09 := "_209000NCP01AK".AA_AK02E3FS52_CH2,
                     I_Alarm10 := "_209000NCP01AK".AA_AK02E3FS53_CH1,
                     I_Alarm11 := "_209000NCP01AK".AA_AK02E3FS53_CH2,
                     I_Alarm12 := "_209000NCP01AK".AA_AK02E3FS54_CH1,
                     I_Alarm13 := "_209000NCP01AK".AA_AK02E3FS54_CH2,
                     I_Alarm14 := "_209000NCP01AK".AD_AK02E3FS50_CH1,
                     I_Alarm15 := "_209000NCP01AK".AD_AK02E3FS51_CH1,
                     I_Alarm16 := "_209000NCP01AK".AD_AK02E3FS51_CH2,
                     I_Alarm17 := "_209000NCP01AK".AD_AK02E3FS52_CH1,
                     I_Alarm18 := "_209000NCP01AK".AD_AK02E3FS52_CH2,
                     I_Alarm19 := "_209000NCP01AK".AD_AK02E3FS53_CH1,
                     I_Alarm20 := "_209000NCP01AK".AD_AK02E3FS53_CH2,
                     I_Alarm21 := "_209000NCP01AK".AD_AK02E3FS54_CH1,
                     I_Alarm22 := "_209000NCP01AK".AD_AK02E3FS54_CH2,
                     I_Alarm23 := "_209000NCP01AK".AC_AK01E1QM6,
                     I_Alarm24 := "_209000NCP01AK".AA_AK01E2FS1,
                     I_Alarm25 := "_209000NCP01AK".AC_AK01E2FS2,
                     I_Alarm26 := "_209000NCP01AK".AC_AK01E2FS3,
                     I_Alarm27 := "_209000NCP01AK".AC_AK01E2FS4,
                     I_Alarm28 := "_209000NCP01AK".AC_AK01E2FS5,
                     I_Alarm29 := "_209000NCP01AK".AC_AK01E2FS6,
                     I_Alarm30 := "_209000NCP01AK".AC_AK01E2FS7,
                     I_Alarm31 := "_209000NCP01AK".AC_AK03EL1,
                     H_AlarmDWord => "_209000NCP01Alarms"."209000NCP01AK_AW1");
   END_IF;
END_REGION

REGION Network 55: **** 9.2 - Alarm DWord**** Alarm To DWord
   // Alarm Word
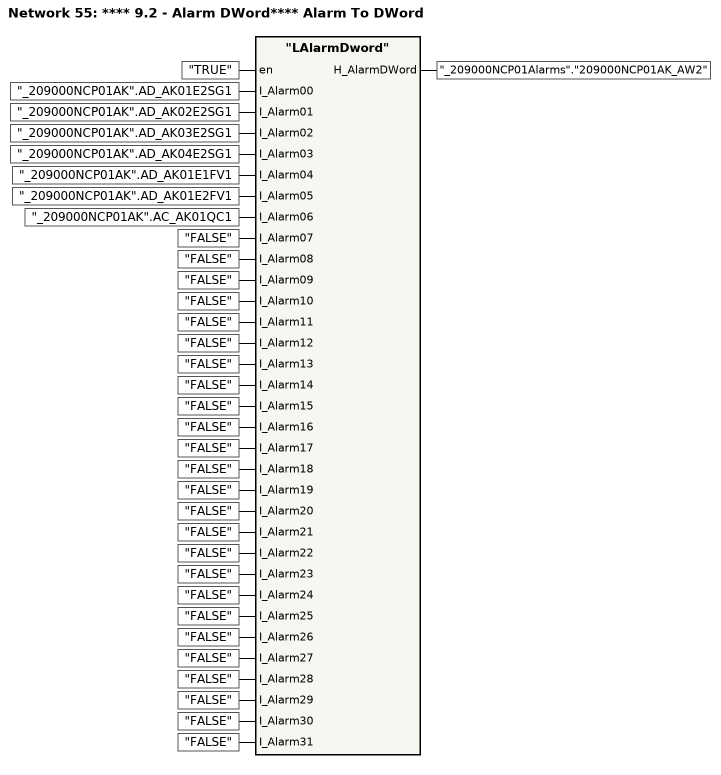
   IF "TRUE" THEN
       "LAlarmDword"(I_Alarm00 := "_209000NCP01AK".AD_AK01E2SG1,
                     I_Alarm01 := "_209000NCP01AK".AD_AK02E2SG1,
                     I_Alarm02 := "_209000NCP01AK".AD_AK03E2SG1,
                     I_Alarm03 := "_209000NCP01AK".AD_AK04E2SG1,
                     I_Alarm04 := "_209000NCP01AK".AD_AK01E1FV1,
                     I_Alarm05 := "_209000NCP01AK".AD_AK01E2FV1,
                     I_Alarm06 := "_209000NCP01AK".AC_AK01QC1,
                     I_Alarm07 := "FALSE",
                     I_Alarm08 := "FALSE",
                     I_Alarm09 := "FALSE",
                     I_Alarm10 := "FALSE",
                     I_Alarm11 := "FALSE",
                     I_Alarm12 := "FALSE",
                     I_Alarm13 := "FALSE",
                     I_Alarm14 := "FALSE",
                     I_Alarm15 := "FALSE",
                     I_Alarm16 := "FALSE",
                     I_Alarm17 := "FALSE",
                     I_Alarm18 := "FALSE",
                     I_Alarm19 := "FALSE",
                     I_Alarm20 := "FALSE",
                     I_Alarm21 := "FALSE",
                     I_Alarm22 := "FALSE",
                     I_Alarm23 := "FALSE",
                     I_Alarm24 := "FALSE",
                     I_Alarm25 := "FALSE",
                     I_Alarm26 := "FALSE",
                     I_Alarm27 := "FALSE",
                     I_Alarm28 := "FALSE",
                     I_Alarm29 := "FALSE",
                     I_Alarm30 := "FALSE",
                     I_Alarm31 := "FALSE",
                     H_AlarmDWord => "_209000NCP01Alarms"."209000NCP01AK_AW2");
   END_IF;
END_REGION
END_FUNCTION
